{attribute 'qualified_only'}
{attribute 'strict'}
{attribute 'to_string'}
TYPE TESTE :
(
	enum_member := 0,
	blarhg
);
END_TYPE

(* stored: Version 1.1.0.1
   DUT TESTE: Id {20554de6-4f9b-4362-90d2-da608912c03d} *)
